(* PLC project Tc2_Utilities.FB_GetRtPerformanceData Demo, tc3-libraries-kb TwinCAT 3.1 *)
(* stored: creationDateTime 2026-05-10T20:00:00, modificationDateTime 2026-05-10T20:00:00 *)

PROGRAM P_Demo_FB_GetRtPerformanceData
  VAR
    fbFB_GetRtPerformanceData : FB_GetRtPerformanceData;  (* Tc2_Utilities.FB_GetRtPerformanceData 实例 *)
    arg_bExecute : BOOL;  (* VAR_INPUT bExecute *)
    arg_bReset : BOOL;  (* VAR_INPUT bReset *)
    arg_tTimeout : TIME;  (* VAR_INPUT tTimeout *)
    arg_sNetId : T_AmsNetId;  (* VAR_INPUT sNetId *)
    arg_bBusy : BOOL;  (* VAR_INPUT bBusy *)
    arg_bError : BOOL;  (* VAR_INPUT bError *)
    arg_nErrorId : UDINT;  (* VAR_INPUT nErrorId *)
    arg_nUsedCpuCount : UDINT;  (* VAR_INPUT nUsedCpuCount *)
    arg_stRtPerformanceData : ARRAY [1..nMaxCpuCount] OF ST_RtPerformanceData;  (* VAR_INPUT stRtPerformanceData *)
  END_VAR

            // ============================================================
// Tc2_Utilities.FB_GetRtPerformanceData 演示程序（FB 实例）
// ============================================================
// 验证步骤：
//   1. 引用 Tc2_Utilities（及依赖类型所在库 Tc2_System 等）
//   2. 编译 + 登录
//   3. 按 doc.md 给 arg_* 赋值
//   4. 在线监视 out_* / io_* 输出
// ============================================================

fbFB_GetRtPerformanceData(
    bExecute := arg_bExecute,
    bReset := arg_bReset,
    tTimeout := arg_tTimeout,
    sNetId := arg_sNetId,
    bBusy := arg_bBusy,
    bError := arg_bError,
    nErrorId := arg_nErrorId,
    nUsedCpuCount := arg_nUsedCpuCount,
    stRtPerformanceData := arg_stRtPerformanceData
);

          
END_PROGRAM
